(* PLC project Unnamed, Unknown Unnamed 1 *)
(* stored: creationDateTime 2025-06-13T17:51:35, modificationDateTime 2025-06-13T18:16:29 *)

PROGRAM part3
  VAR
    state : UINT := 0;
    wait_for_request : UINT := 0;
    wait_for_traffic : UINT := 1;
    slow_cars : UINT := 2;
    ped_xing : UINT := 3;
    all_red : UINT := 4;
    yellow_delay : TIME := T#3s;
    ped_xing_delay : TIME := T#15s;
    all_red_delay : TIME := T#1s;
  END_VAR
  VAR
    car_sensor AT %IX0.0 : BOOL;
    ped_button AT %IX0.1 : BOOL;
    car_red AT %QX0.0 : BOOL;
    car_yellow AT %QX0.1 : BOOL;
    car_green AT %QX0.2 : BOOL;
    ped_red AT %QX0.3 : BOOL;
    ped_green AT %QX0.4 : BOOL;
  END_VAR
  VAR  (* added by the conversion: wires and edge detectors of the diagram *)
    _EQ2_OUT : BOOL;
    _EQ7_OUT : BOOL;
    _EQ10_OUT : BOOL;
    _EQ13_OUT : BOOL;
  END_VAR

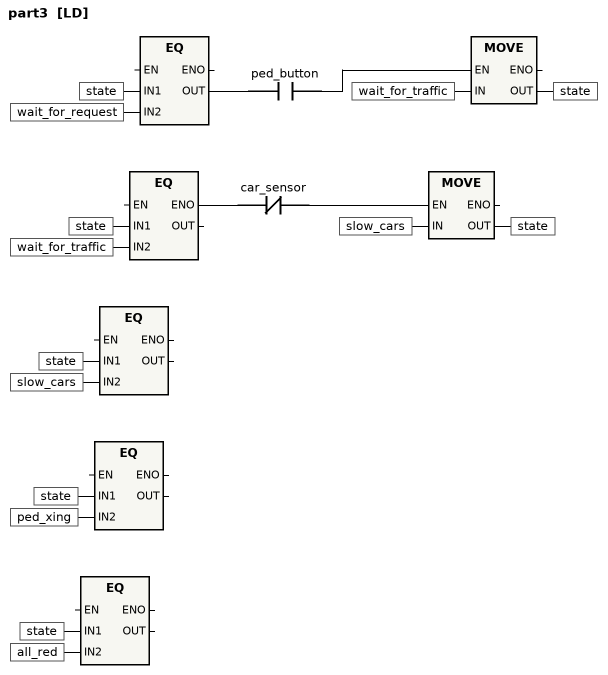
(* LD diagram, written out as Structured Text *)
IF state = wait_for_request AND ped_button THEN state := wait_for_traffic; END_IF;
_EQ2_OUT := state = wait_for_traffic;
IF NOT car_sensor THEN state := slow_cars; END_IF;
_EQ7_OUT := state = slow_cars;
_EQ10_OUT := state = ped_xing;
_EQ13_OUT := state = all_red;
END_PROGRAM

CONFIGURATION Config0
  RESOURCE Res0 ON PLC
    TASK task0(INTERVAL := T#20ms, PRIORITY := 0);
    PROGRAM instance0 WITH task0 : part3;
  END_RESOURCE
END_CONFIGURATION
